PROGRAM MAIN
VAR
	
	bHardwareButton AT %I* : BOOL;
	
	bHmiButton : BOOL;
	
	bMainMotor AT %Q* : BOOL;
	
END_VAR

bMainMotor := bHardwareButton or bHmiButton;

END_PROGRAM

(* stored: Version 1.1.0.1
   POU MAIN: Id {92ad98ed-130f-4aa1-a549-2c21972d48e1}, SpecialFunc None *)
